(* Schneider Machine Expert - Basic project PROJETO_TANK_SUPERVISOR, file version 2.9.0.0 *)
(* ProjectInformations: Name=Novo projeto *)

HARDWARE
  Cpu 0: TM221CE24R
  ModuleExtensionObject 0: TM3TI4D/G
  ModuleExtensionObject 1: TM3AI8/G
  EthernetConfiguration: NetworkName=M221, IpAllocationMode=FixedAddress, IpAddress=0.0.0.0, SubnetMask=0.0.0.0
  SerialLineConfiguration: Baud=Baud19200, Parity=ParityEven, DataBits=DataBits8, StopBits=StopBits1, PhysicalMedium=PhysicalMediumRs485, TransmissionMode=TransmissionModeModbusRtu, SlaveId=1, Addressing=SlaveAddressing
  MastTask: UsePeriodScanMode=false, PeriodScan=100
  FastTask: Period=255
  CpuBehavior: StartingMode=StartAsPreviousState, AutoSaveRamOnEeprom=true, WatchdogPeriod=250

SYMBOLS  (address, symbol, comment, settings)
  %M0       ON_MOTOR
  %M1       OFF_MOTOR
  %M2       MEMAUX_NIVEL
  %M4       EMERG
  %M6       PSV1
  %M10      MOTOR
  %M11      BOMBA_ESCOAMENTO
  %M30      MEMAUX_BOMBA
  %M31      DESLIGA_MOTOR_SOBRECARGA
  %M52      AUT_MANU
  %IW2.0      [Type=Type_4_20mA, Scope=Scope_Customized, Minimum=0, Maximum=100]

POU Novo POU
  (* SectionNumber=1 *)

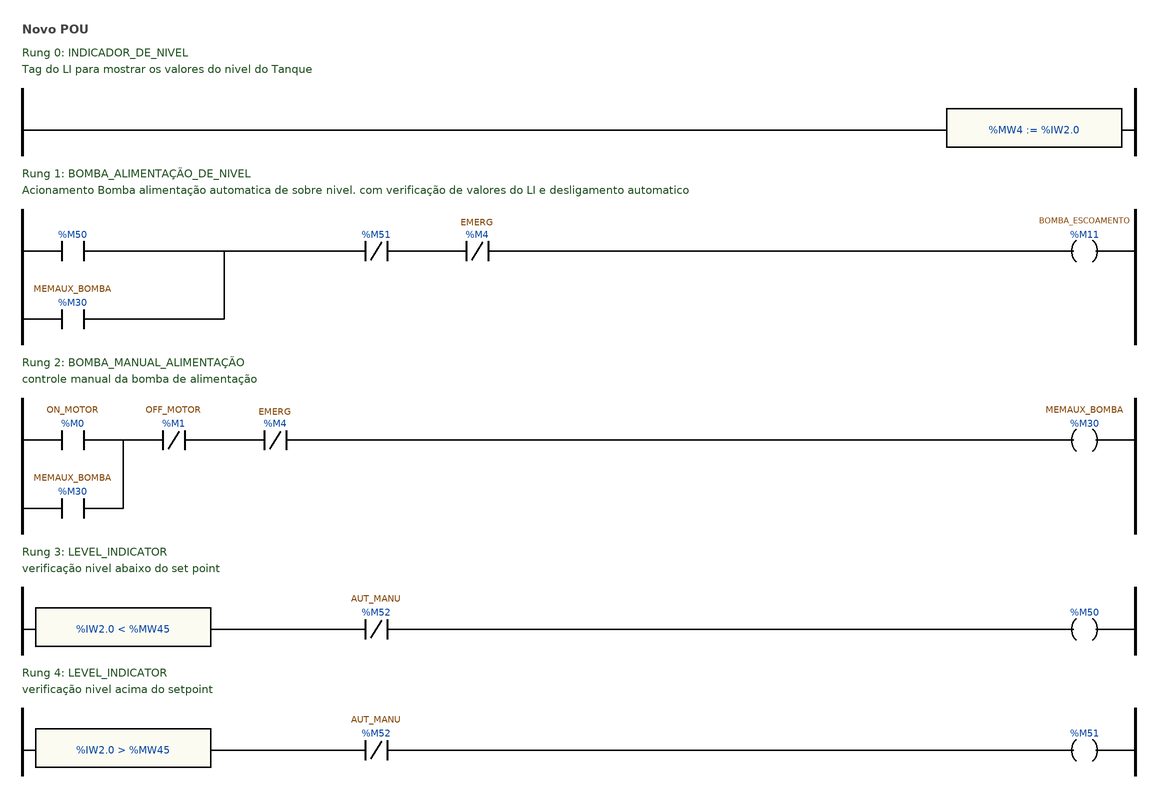

// Rung 0: INDICADOR_DE_NIVEL
// Tag do LI para mostrar os valores do nivel do Tanque
  LD 1
  [ %MW4 := %IW2.0 ]
  // as ST:
  //   %MW4 := %IW2.0;

// Rung 1: BOMBA_ALIMENTAÇÃO_DE_NIVEL
// Acionamento Bomba alimentação automatica de sobre nivel. com verificação de valores do LI e desligamento automatico
  LD %M50
  OR %M30                 (* MEMAUX_BOMBA *)
  ANDN %M51
  ANDN %M4                (* EMERG *)
  ST %M11                 (* BOMBA_ESCOAMENTO *)
  // as ST:
  //   BOMBA_ESCOAMENTO := (%M50 OR MEMAUX_BOMBA) AND NOT %M51 AND NOT EMERG;

// Rung 2: BOMBA_MANUAL_ALIMENTAÇÃO
// controle manual da bomba de alimentação
  LD %M0                  (* ON_MOTOR *)
  OR %M30                 (* MEMAUX_BOMBA *)
  ANDN %M1                (* OFF_MOTOR *)
  ANDN %M4                (* EMERG *)
  ST %M30                 (* MEMAUX_BOMBA *)
  // as ST:
  //   MEMAUX_BOMBA := (ON_MOTOR OR MEMAUX_BOMBA) AND NOT OFF_MOTOR AND NOT EMERG;

// Rung 3: LEVEL_INDICATOR
// verificação nivel abaixo do set point
  LD [ %IW2.0 < %MW45 ]
  ANDN %M52               (* AUT_MANU *)
  ST %M50
  // as ST:
  //   %M50 := %IW2.0 < %MW45 AND NOT AUT_MANU;

// Rung 4: LEVEL_INDICATOR
// verificação nivel acima do setpoint
  LD [ %IW2.0 > %MW45 ]
  ANDN %M52               (* AUT_MANU *)
  ST %M51
  // as ST:
  //   %M51 := %IW2.0 > %MW45 AND NOT AUT_MANU;
